Universal Robots PolyScope program: program2.urp

Program contex (installation=default directory=/ursim/programs createdIn=3.15.8.106339 lastSavedIn=3.15.8.106339 robotSerialNumber=2018359999)
Calibrated DH parameters: a=[0, -0.425, -0.39225, 0, 0, 0]; d=[0.089159, 0, 0, 0.10915, 0.09465, 0.0823]; alpha=[1.570796, 0, 0, 1.570796, -1.570796, 0]; deltaTheta=[0, 0, 0, 0, 0, 0]
Robot Program (runOnlyOnce=false)
  Set DigitalOutput pin=digital_out[0]; digitalValue=1
  Popup Message (haltProgram=false message=Se va a generar un retardo de 5 seg para iniciar un control externo inputType=Text)
  Wait Sleep waitTime=5
  URCap External Control (External Control, FZI Research Center for Information Technology)
